{attribute 'qualified_only'}
{attribute 'strict'}
TYPE E_SafeState :
(
	None,
	Denied, 
	Permit
);
END_TYPE

(* stored: Version 1.1.0.1
   DUT E_SafeState: Id {636b57dc-a143-4e86-99e6-ab587bd0faa0} *)
